FUNCTION_BLOCK Data_Source_Real_2 (* 2 entrys *)
  (* Standard: 61499-2 *)
  (* Version 03-07-12, GASR *)
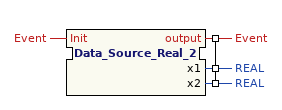
  EVENT_INPUT
    Init;
  END_EVENT
  EVENT_OUTPUT
    output WITH x1, x2;
  END_EVENT
  VAR_OUTPUT
    x1 : REAL;
    x2 : REAL;
  END_VAR
  SERVICE USER/Data_Source_Real_2
    SEQUENCE seq1
      USER.command() -> Data_Source_Real_2.output();
    END_SEQUENCE
  END_SERVICE
END_FUNCTION_BLOCK
